// TIA Portal V19 export
TYPE "LAF_typeRollerEm1Parameters"
// stored: Access Published
   STRUCT
      cm1Vfd205 : "LAF_typeVfdParameters";
   END_STRUCT;
END_TYPE
